// TwinCAT 3 PLC project sample_delivery
// Title: lcls-plc-rix-sample-delivery
// Company: SLAC
// ProjectVersion: 0.0.0
// ProgramVersion: 3.1.4022.7
// libraries:
//   lcls-twincat-sample-delivery, * (SLAC)
//   Tc2_Standard, * (Beckhoff Automation GmbH)
//   Tc2_System, * (Beckhoff Automation GmbH)
//   Tc3_Module, * (Beckhoff Automation GmbH)
// project tree:
//   GVLs/ GVL_SDS.TcGVL
//   / PlcTask.TcTTO, SerialComm.TcTTO
//   POUs/ MAIN.TcPOU, SerialTxRx.TcPOU
// real-time tasks:
//   TASK PlcTask: cycle T#10ms, priority 20, ADS port 350
//   TASK SerialComm: cycle T#5ms, priority 1, ADS port 351
// I/O:
//   DEVICE Device 1 (EtherCAT), AmsNetId 172.21.140.88.2.1
//     Term 1 (EK1200) [EK1200-5000 EtherCAT Power supply (2A E-Bus)]
//       Term 2 (EK1110) [EK1110 EtherCAT extension]
//     Box 3 (EP9128-0021) [EP9128-0021 8x EtherCAT junction]
//       4PV_01 (EP1111) [EP1111-0000 ID-Switch]
//       Box 8 (EP2338-0001) [EP2338-0001 8 Ch. Dig. Input/Output 24V, 0,5A, M8]
//       Term 16 (EP6002-0002) [EP6002-0002 Interface (RS232/422/485)]
//       Term 17 (EP9128-1021) [EP9128-1021 8x EtherCAT junction - Dev A]
//       Term 5 (EP9128-2021) [EP9128-2021 8x EtherCAT junction - Dev B]
//         Solenoid Pair A (EP1111)
//         Solenoid Pair A Digital IO (EP2338-0001)
// variable links:
//   sample_delivery Instance <-> Device 1 (EtherCAT)/Box 3 (EP9128-0021)/Term 16 (EP6002-0002)
//     PlcTask Inputs/GVL_SDS.fb_4PortViciValve_01.fbNporValve.stViciSerial.stComIn/D[0] <-> COM TxPDO-Map Inputs Channel 2/Data In 0
//     PlcTask Inputs/GVL_SDS.fb_4PortViciValve_01.fbNporValve.stViciSerial.stComIn/D[10] <-> COM TxPDO-Map Inputs Channel 2/Data In 10
//     PlcTask Inputs/GVL_SDS.fb_4PortViciValve_01.fbNporValve.stViciSerial.stComIn/D[11] <-> COM TxPDO-Map Inputs Channel 2/Data In 11
//     PlcTask Inputs/GVL_SDS.fb_4PortViciValve_01.fbNporValve.stViciSerial.stComIn/D[12] <-> COM TxPDO-Map Inputs Channel 2/Data In 12
//     PlcTask Inputs/GVL_SDS.fb_4PortViciValve_01.fbNporValve.stViciSerial.stComIn/D[13] <-> COM TxPDO-Map Inputs Channel 2/Data In 13
//     PlcTask Inputs/GVL_SDS.fb_4PortViciValve_01.fbNporValve.stViciSerial.stComIn/D[14] <-> COM TxPDO-Map Inputs Channel 2/Data In 14
//     PlcTask Inputs/GVL_SDS.fb_4PortViciValve_01.fbNporValve.stViciSerial.stComIn/D[15] <-> COM TxPDO-Map Inputs Channel 2/Data In 15
//     PlcTask Inputs/GVL_SDS.fb_4PortViciValve_01.fbNporValve.stViciSerial.stComIn/D[16] <-> COM TxPDO-Map Inputs Channel 2/Data In 16
//     PlcTask Inputs/GVL_SDS.fb_4PortViciValve_01.fbNporValve.stViciSerial.stComIn/D[17] <-> COM TxPDO-Map Inputs Channel 2/Data In 17
//     PlcTask Inputs/GVL_SDS.fb_4PortViciValve_01.fbNporValve.stViciSerial.stComIn/D[18] <-> COM TxPDO-Map Inputs Channel 2/Data In 18
//     PlcTask Inputs/GVL_SDS.fb_4PortViciValve_01.fbNporValve.stViciSerial.stComIn/D[19] <-> COM TxPDO-Map Inputs Channel 2/Data In 19
//     PlcTask Inputs/GVL_SDS.fb_4PortViciValve_01.fbNporValve.stViciSerial.stComIn/D[1] <-> COM TxPDO-Map Inputs Channel 2/Data In 1
//     PlcTask Inputs/GVL_SDS.fb_4PortViciValve_01.fbNporValve.stViciSerial.stComIn/D[20] <-> COM TxPDO-Map Inputs Channel 2/Data In 20
//     PlcTask Inputs/GVL_SDS.fb_4PortViciValve_01.fbNporValve.stViciSerial.stComIn/D[21] <-> COM TxPDO-Map Inputs Channel 2/Data In 21
//     PlcTask Inputs/GVL_SDS.fb_4PortViciValve_01.fbNporValve.stViciSerial.stComIn/D[2] <-> COM TxPDO-Map Inputs Channel 2/Data In 2
//     PlcTask Inputs/GVL_SDS.fb_4PortViciValve_01.fbNporValve.stViciSerial.stComIn/D[3] <-> COM TxPDO-Map Inputs Channel 2/Data In 3
//     PlcTask Inputs/GVL_SDS.fb_4PortViciValve_01.fbNporValve.stViciSerial.stComIn/D[4] <-> COM TxPDO-Map Inputs Channel 2/Data In 4
//     PlcTask Inputs/GVL_SDS.fb_4PortViciValve_01.fbNporValve.stViciSerial.stComIn/D[5] <-> COM TxPDO-Map Inputs Channel 2/Data In 5
//     PlcTask Inputs/GVL_SDS.fb_4PortViciValve_01.fbNporValve.stViciSerial.stComIn/D[6] <-> COM TxPDO-Map Inputs Channel 2/Data In 6
//     PlcTask Inputs/GVL_SDS.fb_4PortViciValve_01.fbNporValve.stViciSerial.stComIn/D[7] <-> COM TxPDO-Map Inputs Channel 2/Data In 7
//     PlcTask Inputs/GVL_SDS.fb_4PortViciValve_01.fbNporValve.stViciSerial.stComIn/D[8] <-> COM TxPDO-Map Inputs Channel 2/Data In 8
//     PlcTask Inputs/GVL_SDS.fb_4PortViciValve_01.fbNporValve.stViciSerial.stComIn/D[9] <-> COM TxPDO-Map Inputs Channel 2/Data In 9
//     PlcTask Inputs/GVL_SDS.fb_4PortViciValve_01.fbNporValve.stViciSerial.stComIn/Status <-> COM TxPDO-Map Inputs Channel 2/Status
//     PlcTask Outputs/GVL_SDS.fb_4PortViciValve_01.fbNporValve.stViciSerial.stComOut/Ctrl <-> COM RxPDO-Map Outputs Channel 2/Ctrl
//     PlcTask Outputs/GVL_SDS.fb_4PortViciValve_01.fbNporValve.stViciSerial.stComOut/D[0] <-> COM RxPDO-Map Outputs Channel 2/Data Out 0
//     PlcTask Outputs/GVL_SDS.fb_4PortViciValve_01.fbNporValve.stViciSerial.stComOut/D[10] <-> COM RxPDO-Map Outputs Channel 2/Data Out 10
//     PlcTask Outputs/GVL_SDS.fb_4PortViciValve_01.fbNporValve.stViciSerial.stComOut/D[11] <-> COM RxPDO-Map Outputs Channel 2/Data Out 11
//     PlcTask Outputs/GVL_SDS.fb_4PortViciValve_01.fbNporValve.stViciSerial.stComOut/D[12] <-> COM RxPDO-Map Outputs Channel 2/Data Out 12
//     PlcTask Outputs/GVL_SDS.fb_4PortViciValve_01.fbNporValve.stViciSerial.stComOut/D[13] <-> COM RxPDO-Map Outputs Channel 2/Data Out 13
//     PlcTask Outputs/GVL_SDS.fb_4PortViciValve_01.fbNporValve.stViciSerial.stComOut/D[14] <-> COM RxPDO-Map Outputs Channel 2/Data Out 14
//     PlcTask Outputs/GVL_SDS.fb_4PortViciValve_01.fbNporValve.stViciSerial.stComOut/D[15] <-> COM RxPDO-Map Outputs Channel 2/Data Out 15
//     PlcTask Outputs/GVL_SDS.fb_4PortViciValve_01.fbNporValve.stViciSerial.stComOut/D[16] <-> COM RxPDO-Map Outputs Channel 2/Data Out 16
//     PlcTask Outputs/GVL_SDS.fb_4PortViciValve_01.fbNporValve.stViciSerial.stComOut/D[17] <-> COM RxPDO-Map Outputs Channel 2/Data Out 17
//     PlcTask Outputs/GVL_SDS.fb_4PortViciValve_01.fbNporValve.stViciSerial.stComOut/D[18] <-> COM RxPDO-Map Outputs Channel 2/Data Out 18
//     PlcTask Outputs/GVL_SDS.fb_4PortViciValve_01.fbNporValve.stViciSerial.stComOut/D[19] <-> COM RxPDO-Map Outputs Channel 2/Data Out 19
//     PlcTask Outputs/GVL_SDS.fb_4PortViciValve_01.fbNporValve.stViciSerial.stComOut/D[1] <-> COM RxPDO-Map Outputs Channel 2/Data Out 1
//     PlcTask Outputs/GVL_SDS.fb_4PortViciValve_01.fbNporValve.stViciSerial.stComOut/D[20] <-> COM RxPDO-Map Outputs Channel 2/Data Out 20
//     PlcTask Outputs/GVL_SDS.fb_4PortViciValve_01.fbNporValve.stViciSerial.stComOut/D[21] <-> COM RxPDO-Map Outputs Channel 2/Data Out 21
//     PlcTask Outputs/GVL_SDS.fb_4PortViciValve_01.fbNporValve.stViciSerial.stComOut/D[2] <-> COM RxPDO-Map Outputs Channel 2/Data Out 2
//     PlcTask Outputs/GVL_SDS.fb_4PortViciValve_01.fbNporValve.stViciSerial.stComOut/D[3] <-> COM RxPDO-Map Outputs Channel 2/Data Out 3
//     PlcTask Outputs/GVL_SDS.fb_4PortViciValve_01.fbNporValve.stViciSerial.stComOut/D[4] <-> COM RxPDO-Map Outputs Channel 2/Data Out 4
//     PlcTask Outputs/GVL_SDS.fb_4PortViciValve_01.fbNporValve.stViciSerial.stComOut/D[5] <-> COM RxPDO-Map Outputs Channel 2/Data Out 5
//     PlcTask Outputs/GVL_SDS.fb_4PortViciValve_01.fbNporValve.stViciSerial.stComOut/D[6] <-> COM RxPDO-Map Outputs Channel 2/Data Out 6
//     PlcTask Outputs/GVL_SDS.fb_4PortViciValve_01.fbNporValve.stViciSerial.stComOut/D[7] <-> COM RxPDO-Map Outputs Channel 2/Data Out 7
//     PlcTask Outputs/GVL_SDS.fb_4PortViciValve_01.fbNporValve.stViciSerial.stComOut/D[8] <-> COM RxPDO-Map Outputs Channel 2/Data Out 8
//     PlcTask Outputs/GVL_SDS.fb_4PortViciValve_01.fbNporValve.stViciSerial.stComOut/D[9] <-> COM RxPDO-Map Outputs Channel 2/Data Out 9
//   sample_delivery Instance <-> Device 1 (EtherCAT)/Box 3 (EP9128-0021)/Term 5 (EP9128-2021)/Solenoid Pair A Digital IO (EP2338-0001)
//     PlcTask Outputs/GVL_SDS.PURGE_VRC_01_CTL <-> Channel 12/Output
//     PlcTask Outputs/GVL_SDS.PURGE_VRC_02_CTL <-> Channel 13/Output
//     PlcTask Outputs/GVL_SDS.SolenoidPairA.q_xDO1 <-> Channel 10/Output
//     PlcTask Outputs/GVL_SDS.SolenoidPairA.q_xDO2 <-> Channel 11/Output

CONFIGURATION sample_delivery
    RESOURCE PLC ON TwinCAT3
        TASK PlcTask(INTERVAL := T#10ms, PRIORITY := 20);
        TASK SerialComm(INTERVAL := T#5ms, PRIORITY := 1);
        PROGRAM MAIN WITH PlcTask : MAIN;
        PROGRAM SerialTxRx WITH SerialComm : SerialTxRx;
    END_RESOURCE
END_CONFIGURATION

// ---- GVLs/GVL_SDS.TcGVL
VAR_GLOBAL
    // 4 Port Valve
    {attribute 'pytmc' := 'pv: CRIX:SDS:VICI:01'}
    {attribute 'TcLinkTo' := '.fbNporValve.stViciSerial.stComIn.Status := TIIB[Term 16 (EP6002-0002)]^COM TxPDO-Map Inputs Channel 2^Status;
                              .fbNporValve.stViciSerial.stComOut.Ctrl := TIIB[Term 16 (EP6002-0002)]^COM RxPDO-Map Outputs Channel 2^Ctrl;
                              .fbNporValve.stViciSerial.stComIn.D[0] := TIIB[Term 16 (EP6002-0002)]^COM TxPDO-Map Inputs Channel 2^Data In 0;
                              .fbNporValve.stViciSerial.stComIn.D[1] := TIIB[Term 16 (EP6002-0002)]^COM TxPDO-Map Inputs Channel 2^Data In 1;
                              .fbNporValve.stViciSerial.stComIn.D[2] := TIIB[Term 16 (EP6002-0002)]^COM TxPDO-Map Inputs Channel 2^Data In 2;
                              .fbNporValve.stViciSerial.stComIn.D[3] := TIIB[Term 16 (EP6002-0002)]^COM TxPDO-Map Inputs Channel 2^Data In 3;
                              .fbNporValve.stViciSerial.stComIn.D[4] := TIIB[Term 16 (EP6002-0002)]^COM TxPDO-Map Inputs Channel 2^Data In 4;
                              .fbNporValve.stViciSerial.stComIn.D[5] := TIIB[Term 16 (EP6002-0002)]^COM TxPDO-Map Inputs Channel 2^Data In 5;
                              .fbNporValve.stViciSerial.stComIn.D[6] := TIIB[Term 16 (EP6002-0002)]^COM TxPDO-Map Inputs Channel 2^Data In 6;
                              .fbNporValve.stViciSerial.stComIn.D[7] := TIIB[Term 16 (EP6002-0002)]^COM TxPDO-Map Inputs Channel 2^Data In 7;
                              .fbNporValve.stViciSerial.stComIn.D[8] := TIIB[Term 16 (EP6002-0002)]^COM TxPDO-Map Inputs Channel 2^Data In 8;
                              .fbNporValve.stViciSerial.stComIn.D[9] := TIIB[Term 16 (EP6002-0002)]^COM TxPDO-Map Inputs Channel 2^Data In 9;
                              .fbNporValve.stViciSerial.stComIn.D[10] := TIIB[Term 16 (EP6002-0002)]^COM TxPDO-Map Inputs Channel 2^Data In 10;
                              .fbNporValve.stViciSerial.stComIn.D[11] := TIIB[Term 16 (EP6002-0002)]^COM TxPDO-Map Inputs Channel 2^Data In 11;
                              .fbNporValve.stViciSerial.stComIn.D[12] := TIIB[Term 16 (EP6002-0002)]^COM TxPDO-Map Inputs Channel 2^Data In 12;
                              .fbNporValve.stViciSerial.stComIn.D[13] := TIIB[Term 16 (EP6002-0002)]^COM TxPDO-Map Inputs Channel 2^Data In 13;
                              .fbNporValve.stViciSerial.stComIn.D[14] := TIIB[Term 16 (EP6002-0002)]^COM TxPDO-Map Inputs Channel 2^Data In 14;
                              .fbNporValve.stViciSerial.stComIn.D[15] := TIIB[Term 16 (EP6002-0002)]^COM TxPDO-Map Inputs Channel 2^Data In 15;
                              .fbNporValve.stViciSerial.stComIn.D[16] := TIIB[Term 16 (EP6002-0002)]^COM TxPDO-Map Inputs Channel 2^Data In 16;
                              .fbNporValve.stViciSerial.stComIn.D[17] := TIIB[Term 16 (EP6002-0002)]^COM TxPDO-Map Inputs Channel 2^Data In 17;
                              .fbNporValve.stViciSerial.stComIn.D[18] := TIIB[Term 16 (EP6002-0002)]^COM TxPDO-Map Inputs Channel 2^Data In 18;
                              .fbNporValve.stViciSerial.stComIn.D[19] := TIIB[Term 16 (EP6002-0002)]^COM TxPDO-Map Inputs Channel 2^Data In 19;
                              .fbNporValve.stViciSerial.stComIn.D[20] := TIIB[Term 16 (EP6002-0002)]^COM TxPDO-Map Inputs Channel 2^Data In 20;
                              .fbNporValve.stViciSerial.stComIn.D[21] := TIIB[Term 16 (EP6002-0002)]^COM TxPDO-Map Inputs Channel 2^Data In 21;
                              .fbNporValve.stViciSerial.stComOut.D[0] := TIIB[Term 16 (EP6002-0002)]^COM RxPDO-Map Outputs Channel 2^Data Out 0;
                              .fbNporValve.stViciSerial.stComOut.D[1] := TIIB[Term 16 (EP6002-0002)]^COM RxPDO-Map Outputs Channel 2^Data Out 1;
                              .fbNporValve.stViciSerial.stComOut.D[2] := TIIB[Term 16 (EP6002-0002)]^COM RxPDO-Map Outputs Channel 2^Data Out 2;
                              .fbNporValve.stViciSerial.stComOut.D[3] := TIIB[Term 16 (EP6002-0002)]^COM RxPDO-Map Outputs Channel 2^Data Out 3;
                              .fbNporValve.stViciSerial.stComOut.D[4] := TIIB[Term 16 (EP6002-0002)]^COM RxPDO-Map Outputs Channel 2^Data Out 4;
                              .fbNporValve.stViciSerial.stComOut.D[5] := TIIB[Term 16 (EP6002-0002)]^COM RxPDO-Map Outputs Channel 2^Data Out 5;
                              .fbNporValve.stViciSerial.stComOut.D[6] := TIIB[Term 16 (EP6002-0002)]^COM RxPDO-Map Outputs Channel 2^Data Out 6;
                              .fbNporValve.stViciSerial.stComOut.D[7] := TIIB[Term 16 (EP6002-0002)]^COM RxPDO-Map Outputs Channel 2^Data Out 7;
                              .fbNporValve.stViciSerial.stComOut.D[8] := TIIB[Term 16 (EP6002-0002)]^COM RxPDO-Map Outputs Channel 2^Data Out 8;
                              .fbNporValve.stViciSerial.stComOut.D[9] := TIIB[Term 16 (EP6002-0002)]^COM RxPDO-Map Outputs Channel 2^Data Out 9;
                              .fbNporValve.stViciSerial.stComOut.D[10] := TIIB[Term 16 (EP6002-0002)]^COM RxPDO-Map Outputs Channel 2^Data Out 10;
                              .fbNporValve.stViciSerial.stComOut.D[11] := TIIB[Term 16 (EP6002-0002)]^COM RxPDO-Map Outputs Channel 2^Data Out 11;
                              .fbNporValve.stViciSerial.stComOut.D[12] := TIIB[Term 16 (EP6002-0002)]^COM RxPDO-Map Outputs Channel 2^Data Out 12;
                              .fbNporValve.stViciSerial.stComOut.D[13] := TIIB[Term 16 (EP6002-0002)]^COM RxPDO-Map Outputs Channel 2^Data Out 13;
                              .fbNporValve.stViciSerial.stComOut.D[14] := TIIB[Term 16 (EP6002-0002)]^COM RxPDO-Map Outputs Channel 2^Data Out 14;
                              .fbNporValve.stViciSerial.stComOut.D[15] := TIIB[Term 16 (EP6002-0002)]^COM RxPDO-Map Outputs Channel 2^Data Out 15;
                              .fbNporValve.stViciSerial.stComOut.D[16] := TIIB[Term 16 (EP6002-0002)]^COM RxPDO-Map Outputs Channel 2^Data Out 16;
                              .fbNporValve.stViciSerial.stComOut.D[17] := TIIB[Term 16 (EP6002-0002)]^COM RxPDO-Map Outputs Channel 2^Data Out 17;
                              .fbNporValve.stViciSerial.stComOut.D[18] := TIIB[Term 16 (EP6002-0002)]^COM RxPDO-Map Outputs Channel 2^Data Out 18;
                              .fbNporValve.stViciSerial.stComOut.D[19] := TIIB[Term 16 (EP6002-0002)]^COM RxPDO-Map Outputs Channel 2^Data Out 19;
                              .fbNporValve.stViciSerial.stComOut.D[20] := TIIB[Term 16 (EP6002-0002)]^COM RxPDO-Map Outputs Channel 2^Data Out 20;
                              .fbNporValve.stViciSerial.stComOut.D[21] := TIIB[Term 16 (EP6002-0002)]^COM RxPDO-Map Outputs Channel 2^Data Out 21;

    '}

    fb_4PortViciValve_01 : FB_4PortViciValve;

    {attribute 'pytmc' := 'pv: RIX:SDS:SPR:A'}
    {attribute 'TcLinkTo' := '.q_xDO1 := TIIB[Solenoid Pair A Digital IO (EP2338-0001)]^Channel 10^Output;
                          .q_xDO2 := TIIB[Solenoid Pair A Digital IO (EP2338-0001)]^Channel 11^Output;
    '}
    SolenoidPairA : FB_SolenoidPair;

    // Purge Valves
    {attribute 'pytmc' := 'pv: RIX:SDS:SPR:PURGE:A'}
    {attribute 'TcLinkTo' := 'TIIB[Solenoid Pair A Digital IO (EP2338-0001)]^Channel 12^Output'}
    PURGE_VRC_01_CTL AT%Q* : BOOL;

    {attribute 'pytmc' := 'pv: RIX:SDS:SPR:PURGE:B'}
    {attribute 'TcLinkTo' := 'TIIB[Solenoid Pair A Digital IO (EP2338-0001)]^Channel 13^Output'}
    PURGE_VRC_02_CTL AT%Q* : BOOL;



END_VAR

// ---- POUs/MAIN.TcPOU
PROGRAM MAIN
VAR
END_VAR

SolenoidPairA();

fb_4PortViciValve_01(iAdress:=1);

(* Following execution of all the programs, set the first pass false *)
g_xFirstPass := FALSE;

END_PROGRAM

// ---- POUs/SerialTxRx.TcPOU
PROGRAM SerialTxRx
VAR
END_VAR

(*M3SelectorA.SerialComm();
M3SelectorB.SerialComm();
M3SelectorC.SerialComm();
M3SelectorD.SerialComm();

PCMA.SerialComm();
PCMB.SerialComm();
PCMC.SerialComm();
PCMD.SerialComm();
*)

END_PROGRAM
